{attribute 'GeneratedUsingTerminal: KL2751'}
{attribute addProperty BoxType "KL2751"}
{attribute addProperty Id "Channel_1AT %Q*Channel_6576A6810"}
{attribute addProperty CRC "1632160004"}
{attribute addProperty Size "0"}
TYPE KL2751_6148C904 :
STRUCT
	{attribute addProperty Name "Channel_1"}
	Channel_1 : Channel_6576A681;
END_STRUCT
END_TYPE

(* stored: Version 1.2.0.0, ProductVersion 3.1.4024.9
   DUT KL2751_6148C904: Id {36ae6527-8ec8-46ff-8b12-c9bebaa725ca} *)
